// TwinCAT 3 PLC project Untitled1
// ProgramVersion: 3.1.4022.1
// libraries:
//   Tc2_Standard, * (Beckhoff Automation GmbH)
//   Tc2_System, * (Beckhoff Automation GmbH)
//   Tc2_TcpIp, * (Beckhoff Automation GmbH)
//   Tc3_Module, * (Beckhoff Automation GmbH)
// project tree:
//   / GlobalTextList.TcGTLO, PlcTask.TcTTO, Visualization Manager.TcVMO (not stored)
//   POUs/ automatic.TcPOU, beamer.TcPOU, hysterisis.TcPOU, lichten.TcPOU, MAIN_test.TcPOU, MAIN.TcPOU
//   VISUs/ Visualization.TcVIS

CONFIGURATION Untitled1
    RESOURCE PLC ON TwinCAT3
        TASK PlcTask(INTERVAL := T#10ms, PRIORITY := 20);
        PROGRAM MAIN WITH PlcTask : MAIN;
    END_RESOURCE
END_CONFIGURATION

// ---- POUs/MAIN.TcPOU
PROGRAM MAIN
VAR
	Motion_1	AT %I* 	: BOOL;
	Motion_2 	AT %I*	: BOOL;
	Relay_1 	AT %Q*	: BOOL;
	Relay_2 	AT %Q*	: BOOL;	
	vDruk_1				: BOOL;
	vDruk_2				: BOOL;	
	Druk_1		AT %I*	: BOOL;
	Druk_2		AT %I*	: BOOL;	
	LDR_1		AT %I* 	: INT;
	LDR_2		AT %I* 	: INT;
	LDR_3		AT %I* 	: INT;
	LDR_4		AT %I* 	: INT;
	TOF1			: TOF;
	F_TRIG1			: F_Trig;
	
	lichten_1		: lichten;
	lichten_2		: lichten;
	TOF2, TOF3		: TOF;
	F_TOF2, F_TOF3	: F_Trig;

	Inschakelen_1	: BOOL;
	ENABLE			: BOOL;
	TON1: TON;
	licht1: BOOL;
	licht2: BOOL;
	Aanwezigheid: TOF;
	fAanwezigheid: F_TRIG;
	Debug: BOOL;
END_VAR

IF Debug THEN
	lichten_1(
		Toggle:= vDruk_1 OR Druk_1, 
		ON:= , 
		OFF:= fAanwezigheid.Q, 
		Enable:= NOT(lichten_2.Q), 
		lamp=> , 
		Q=> Relay_1);
		
	lichten_2(
		Toggle:= vDruk_2 OR Druk_2, 
		ON:= , 
		OFF:= fAanwezigheid.Q, 
		Enable:= NOT(lichten_1.Q), 
		lamp=> , 
		Q=> Relay_2);
		
	Aanwezigheid(IN := Motion_1 OR Motion_2, PT := T#5S);
	fAanwezigheid(CLK:= Aanwezigheid.Q);
ELSE
	Relay_1 := Druk_1 OR vDruk_1;
	Relay_2 := Druk_2 OR vDruk_2;
END_IF

END_PROGRAM

// ---- POUs/lichten.TcPOU
FUNCTION_BLOCK lichten
VAR_INPUT
	Toggle 	: BOOL;
	ON 		: BOOL;
	OFF		: BOOL;
	Enable 	: BOOL;
END_VAR
VAR_OUTPUT
	lamp 	: BOOL;
	Q		: BOOL;	// puls 100ms
END_VAR
VAR
	pLamp	: BOOL;
	pToggle : BOOL;
	pON 	: BOOL;
	pOFF	: BOOL;
	puls	: TP;
END_VAR

pLamp := lamp;

IF Toggle THEN pToggle := TRUE; END_IF
IF ON THEN pON := TRUE; END_IF
IF OFF THEN pOFF := TRUE; END_IF

IF Enable AND NOT(puls.Q) THEN
	IF pON THEN lamp := TRUE; pON := FALSE;
	ELSIF pOFF THEN lamp := FALSE; pOFF := FALSE;
	ELSIF pToggle THEN lamp := NOT lamp; pToggle := FALSE;
	END_IF;
END_IF

IF lamp <> pLamp THEN puls.IN := TRUE; ELSE puls.IN := FALSE; END_IF

puls(PT := T#250MS, Q => Q);

END_FUNCTION_BLOCK

// ---- POUs/automatic.TcPOU
FUNCTION_BLOCK automatic
VAR_INPUT
	LDR1, LDR2		: INT;
	LDR_threshold	: INT;
	LDR_duty		: INT;
	motion			: BOOL;
END_VAR
VAR_OUTPUT
	fQ	: BOOL;
	rQ	: BOOL;
END_VAR
VAR
	Motion_ton	: TON;
	Motion_tof	: TOF;
	LDR_tof		: TOF;
	fTRIG: F_TRIG;
	rTRIG: R_TRIG;
	LDR_low: BOOL;
	hys1: hysterisis;
	hys2: hysterisis;
END_VAR

Motion_ton( IN := motion, PT := T#1S );
Motion_tof( IN := Motion_ton.Q, PT := T#5M );

hys1(IN:= LDR1, thresh:= LDR_threshold, variatie:= LDR_duty );
hys2(IN:= LDR2, thresh:= LDR_threshold, variatie:= LDR_duty );

IF Motion_tof.Q THEN
	IF (hys1.UP) AND NOT(hys2.UP) ) THEN
	IF (LDR1 < LDR_threshold) OR (LDR2 < LDR_threshold) THEN
		LDR_low := TRUE;
	ELSIF (LDR1 > LDR_threshold) OR (LDR2 < LDR_threshold)
		LDR_tof.IN := FALSE;
	END_IF
ELSE
	LDR_tof.IN := FALSE;
END_IF

LDR_tof( PT := T#1M );

fTRIG(CLK := LDR_tof.Q ,Q=> );
rTRIG(CLK := LDR_tof.Q ,Q=> );

END_FUNCTION_BLOCK

// ---- POUs/hysterisis.TcPOU
FUNCTION_BLOCK hysterisis
VAR_INPUT
	IN		: INT;
	thresh	: INT;
	variatie: INT;
END_VAR
VAR_OUTPUT
	UP		: BOOL;
END_VAR
VAR
END_VAR

IF IN > (thresh + variatie) THEN
	UP := TRUE;
ELSIF IN < (thresh - variatie) THEN
	UP := FALSE;
END_IF

END_FUNCTION_BLOCK

// ---- POUs/beamer.TcPOU
PROGRAM beamer

VAR
	fbsocketsend: FB_SocketSend;
	bconnect AT %I* : BOOL;
	test : int;
	clientserver: FB_ClientServerConnection;
	Beamerstand: LINT;
	BeamerAANKNOP: BOOL;
	BeamerUITKNOP: BOOL;
	bENABLE: BOOL;
END_VAR

VAR_INPUT
	nMode           	: DWORD := 16#8000000;
	BeamerON    		: LINT := 16#020000000002;
	BeamerOFF 			: LINT := 16#020100000003;
	beamerINPUTCHANGE 	: LINT :=16#020300000201060E;
	sSrvNetId       	: T_AmsNetId := '5.52.70.129.1.1';
	sRemoteHost     	: STRING(15) := '192.168.1.100';
    nRemotePort     	: UDINT := 7142;
    bExecute         	: BOOL;
    tTimeout            : TIME := T#45S;
	tReconnect      	: TIME := T#45S;(*!!!*)

	//socketsend       
    cbLen           : UDINT;                        
    pSrc            : DWORD;       
END_VAR  

VAR_OUTPUT
	bBusy           : BOOL;
    bError          : BOOL;
    nErrId          : UDINT;
	nErrId2         : UDINT;
    hSocket        	: T_HSOCKET;
	eState          : E_SocketConnectionState := eSOCKET_DISCONNECTED;
END_VAR

clientserver(
	sSrvNetID:= '', 
	nMode:=CONNECT_MODE_ENABLEDBG , 
	sRemoteHost:= sremoteHost , 
	nRemotePort:= nremoteport, 
	bEnable:= TRUE, 
	tReconnect:= tReconnect, 
	bBusy=> , 
	bError=> ,
	nErrId=>nErrId , 
	hSocket=>hsocket , 
	eState=> eState
);
	
IF 		BeamerUITKNOP = TRUE THEN Beamerstand := BeamerOFF;
ELSIF 	BeamerAANKNOP = TRUE THEN Beamerstand := BeamerON;
ELSE	Beamerstand := 0; 	 END_IF

IF NOT clientserver.bBusy AND clientserver.bEnable AND NOT clientserver.bError THEN
	fbsocketsend(
		sSrvNetId:='' , 
		hSocket:= clientserver.hSocket, 
		cbLen:= 50, 
		pSrc:= ADR(Beamerstand), 
		bExecute:= BeamerUITKNOP OR BeamerAANKNOP , 
		tTimeout:=tTimeout , 
		bBusy=> bBusy , 
		bError=> bError, 
		nErrId=> nErrId2
	);
END_IF

END_PROGRAM

// ---- POUs/MAIN_test.TcPOU
PROGRAM MAIN_test
VAR
	Motion_1	AT %I* 	: BOOL;
	Motion_2 	AT %I*	: BOOL;
	Relay_1 	AT %Q*	: BOOL;
	Relay_2 	AT %Q*	: BOOL;	
	vDruk_1				: BOOL;
	vDruk_2				: BOOL;	
	Druk_1		AT %I*	: BOOL;
	Druk_2		AT %I*	: BOOL;	
	LDR_1		AT %I* 	: INT;
	LDR_2		AT %I* 	: INT;
	LDR_3		AT %I* 	: INT;
	LDR_4		AT %I* 	: INT;
	
	TOF1			: TOF;
	F_TRIG1			: F_Trig;
	
	lichten_1		: lichten;
	lichten_2		: lichten;
	TOF2, TOF3		: TOF;
	F_TOF2, F_TOF3	: F_Trig;

	Inschakelen_1	: BOOL;
	ENABLE			: BOOL;
	TON1			: TON;
	
	automatic_1: automatic;
	automatic_2: automatic;
	auto_ON : BOOL;
END_VAR

automatic_1(	LDR1:= LDR_1, LDR2:= LDR_2, LDR_threshold:= 500, motion:= Motion_1 );
automatic_2(	LDR1:= LDR_3, LDR2:= LDR_4, LDR_threshold:= 500, motion:= Motion_2 );



IF druk_2 THEN auto_ON := NOT auto_ON; END_IF
				
IF auto_ON THEN
	lichten_1.ON:= automatic_1.ON;
	lichten_1.OFF:= automatic_1.OFF;
	lichten_2.ON:= automatic_2.ON;
	lichten_2.OFF := automatic_2.OFF;
ELSE
	lichten_1.ON:= FALSE;
	lichten_1.OFF:= FALSE;
	lichten_2.ON:= FALSE;
	lichten_2.OFF := FALSE;
END_IF
				
lichten_1(	toggle:= vDruk_1 OR Druk_1, 
			 Q=> Relay_1 );

lichten_2(	toggle:= vDruk_2 OR Druk_1, 
			ON:= automatic_2.ON, OFF:= automatic_2.OFF, Q=> Relay_2 );
			
beamer();

END_PROGRAM

// ---- GlobalTextList.TcGTLO
TEXTLIST GlobalTextList
  584 = '%d'
  90 = 'druk'
  64 = 'ingang2'
END_TEXTLIST

// ---- VISUs/Visualization.TcVIS
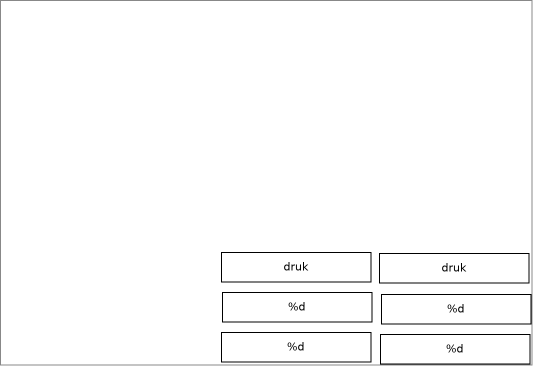
VISUALIZATION Visualization  // 533x366
    Rectangle (221,252 150x30), "druk", colour toggle: MAIN.lichten_1.lamp
        tap MAIN.vDruk_1
    Rectangle (379,253 150x30), "druk", colour toggle: MAIN.lichten_2.lamp
        tap MAIN.vDruk_2
    Rectangle (222,292 150x30), "%d", text variable: MAIN.LDR_1
    Rectangle (381,294 150x30), "%d", text variable: MAIN.LDR_2
    Rectangle (221,332 150x30), "%d", text variable: MAIN.LDR_3
    Rectangle (380,334 150x30), "%d", text variable: MAIN.LDR_4
END_VISUALIZATION
